{attribute 'enable_dynamic_creation'}
FUNCTION_BLOCK FB_CleaningBrush EXTENDS FB_TargetBase
VAR_INPUT
END_VAR
VAR_OUTPUT
END_VAR

VAR
	rMargin  : REAL;
END_VAR

METHOD FB_init : BOOL
VAR_INPUT
	bInitRetains : BOOL; // if TRUE, the retain variables are initialized (warm start / cold start)
	bInCopyCode : BOOL;  // if TRUE, the instance afterwards gets moved into the copy code (online change)
END_VAR
eObjectType := E_ObjectType.OBJECTTYPE_CleaningBrush;
eObjectGroup := E_ObjectGroup.OBJECTGROUP_Target;
END_METHOD

METHOD M_GetAllProps : ERRORID
VAR_INPUT
	refCmdData : REFERENCE TO  ST_CmdData;
END_VAR
SUPER^.M_GetAllProps(refCmdData);
nCurrentPropIndex := nCurrentPropIndex + 1;
refCmdData.n32Data[nCurrentPropIndex] := REAL_TO_DINT(rMargin);
END_METHOD

{attribute 'object_name' := 'M_SetAllProps'}
METHOD M_SetAllProps : ERRORID
VAR_INPUT
	refCmdData	: REFERENCE TO ST_CmdData;
END_VAR
M_SetAllProps := SUPER^.M_SetAllProps(refCmdData);

IF M_SetAllProps > 0 THEN
	RETURN;
END_IF

nCurrentPropIndex := nCurrentPropIndex + 1;
rMargin := DINT_TO_REAL(refCmdData.n32Data[nCurrentPropIndex]);
nNoOfProps := nCurrentPropIndex + 1;
END_METHOD

PROPERTY P_rMargin : REAL
GET
P_rMargin := rMargin;
END_GET
END_PROPERTY

END_FUNCTION_BLOCK

(* stored: Version 1.1.0.1, ProductVersion 3.1.4024.6
   POU FB_CleaningBrush: Id {f861d869-f23d-4f55-afaa-062e260f8370}, SpecialFunc None
   Method FB_init: Id {f0576d75-c9f8-4e7a-adcb-b6267f89f0c5}
   Method M_GetAllProps: Id {4ddb9170-d3df-4029-9f18-edc7d4867c6e}
   Method M_SetAllProps: Id {ee8467a6-4eb3-49fe-b7d1-c765cb28dcbe}
   Property P_rMargin: Id {8d4bd7bf-87ee-43b0-8cc1-c78734bab539}
   Get Get: Id {452c587f-7bef-4614-9e0d-3ff0f9b2aa99} *)
